(* PLC project button, Dassault Systèmes ControlBuild 2024x *)
(* stored: creationDateTime 2023-10-03T11:13:58-01:00 *)

FUNCTION_BLOCK tri_chain.button
  VAR_OUTPUT
    output : BOOL := false;
  END_VAR
  VAR
    user_PushButton : BOOL := false;
    time2reach : BOOL := false;
  END_VAR
  VAR CONSTANT
    pulse_type : BOOL := false;
    pulseDuration : REAL := 2.0;
  END_VAR


ACTION C_source_code:
/* ----------------------------------------------------------------	*/
/* Type : Model of Operative Behaviour					*/
/* Category :  Sensors							*/
/* Author : Dassault Systemes						*/
/* Update date : June 2018							*/
/* ----------------------------------------------------------------	*/
if pulse_type 
	{
	if user_PushButton
		{
		if(timeNow >= time2reach) user_PushButton=0;
		}
	else
		{
		time2reach=timeNow+(pulseDuration * 1000000);
		}
	output=user_PushButton;
	}
else
	{
	output=user_PushButton;
	}
END_ACTION
END_FUNCTION_BLOCK
